FUNCTION_BLOCK FB_SL3K4
VAR CONSTANT
    nActiveMotorCount    : UINT := 4;
END_VAR
VAR_IN_OUT
	astMotionStage   : ARRAY[1..MotionConstants.MAX_STATE_MOTORS] OF ST_MotionStage;
	astChanParam     : ARRAY[1..MotionConstants.MAX_STATE_MOTORS] OF ST_MCS2ChanParameter;
    fbArbiter        : FB_Arbiter;
    fbFFHWO          : FB_HardwareFFOutput;
END_VAR
VAR_INPUT
	{attribute 'hide'}
    bFileReaderBusy      : BOOL;
	{attribute 'hide'}
    bFileReaderError     : BOOL;
	{attribute 'hide'}
    sTransitionKey       : STRING;
	{attribute 'hide'}
    bEnableDriftCheck    : BOOL := TRUE;
	{attribute 'hide'}
    fDriftTolerance      : LREAL := 0.003;
	{attribute 'hide'}
    bEnableBeamParams    : BOOL := TRUE;
    bReadDBNow           : BOOL;

END_VAR
VAR
    {attribute 'hide'}
    fbPerMotorFFO        : FB_PerMotorFFOND;
    {attribute 'hide'}
    fbMiscStatesErrorFFO : FB_MiscStatesErrorFFO;
    {attribute 'hide'}
    ffDriftFFO           : FB_FastFault;
    {attribute 'hide'}
    ffProgrammerError    : FB_FastFault;
    {attribute 'hide'}
    fbSL3K4BPTM          : FB_SL3K4BPTM;
    {attribute 'hide'}
    fbMotionClearAsserts : FB_MotionClearAsserts;
	
    {attribute 'pytmc' := '
        pv: STATE
        io: io
        field: DESC SL3K4 state
    '}
    eSL3K4State	: UINT := E_SL3K4State.NORMAL;
	
    {attribute 'pytmc' := 'pv: STATE'}
    stPMPSEpicsToPlc     : ST_StatePMPSEpicsToPlc;
	
    {attribute 'hide'}
    ePrevState            : E_SL3K4State := E_SL3K4State.NORMAL;

    {attribute 'hide'}
    abBladeEnable        : ARRAY[1..MotionConstants.MAX_STATE_MOTORS] OF BOOL;
    {attribute 'hide'}
    stMaintenanceGoal    : ST_DbStateParams;
    {attribute 'hide'}
    stNormalGoal         : ST_DbStateParams;
    {attribute 'hide'}
    stTransitionGoal     : ST_DbStateParams;
    {attribute 'hide'}
    bDBStatesLoaded      : BOOL := FALSE;
    {attribute 'hide'}
    bSafeToMove          : BOOL;
    {attribute 'hide'}
    bLocked              : BOOL;
    {attribute 'hide'}
    bMaintenanceActive   : BOOL;
    {attribute 'hide'}
    bProgrammerError     : BOOL;
    {attribute 'hide'}
    sStatusMsg           : STRING;
    {attribute 'hide'}
    bAnybladeError       : BOOL;
    {attribute 'hide'}
    bArbiterError        : BOOL;
    {attribute 'hide'}
    nBlades              : UINT;
    {attribute 'hide'}
    fbSL3K4ReadPMPSDB    : FB_SL3K4ReadPMPSDB;
    {attribute 'hide'}
    sDeviceName          : STRING := 'SL3K4';
    {attribute 'hide'}
    stGoalParams         : ST_DbStateParams;
    {attribute 'hide'}
    stTransParams        : ST_DbStateParams;
    {attribute 'hide'}
    bDBReloadRequested   : BOOL := TRUE;
    {attribute 'hide'}
    bDBReloadNow         : BOOL;
    {attribute 'hide'}
    bReadNow             : BOOL;
    {attribute 'hide'}
    bDone                : BOOL;
    {attribute 'hide'}
    bDriftFF             : BOOL;
    {attribute 'hide'}
    bLastTransAuth       : BOOL;
    {attribute 'hide'}
    bEnable              : BOOL;
    {attribute 'hide'}
    tArbiterTimeout      : TIME := T#3s;
    {attribute 'hide'}
    bMoveOnArbiterTimeout: BOOL := TRUE;
    {attribute 'hide'}
    bResetBPTMTimeout    : BOOL;
    {attribute 'hide'}
    bRetry               : BOOL;
    {attribute 'hide'}
    bAtState             : BOOL;
    {attribute 'hide'}
    bInternalAuth        : BOOL;
    {attribute 'hide'}
    bArbiterTimeout      : BOOL;
    arfDrift               : ARRAY[1..nActiveMotorCount] OF LREAL;
    {attribute 'hide'}
    allAxesIdle          : BOOL;
    {attribute 'hide'}
    axis                 : INT;
    {attribute 'hide'}
    i                    : DINT;
    {attribute 'hide'}
    bIsMaintenance       : BOOL;
    {attribute 'hide'}
    bGoalIsNormal        : BOOL;
    {attribute 'hide'}
    bFoundTransition     : BOOL;
    {attribute 'hide'}
    bFoundGoal           : BOOL;
    {attribute 'hide'}
    fbLogger             : FB_LogMessage := (eSubsystem:=E_SubSystem.MOTION);
    {attribute 'hide'}
    eSevr                : LCLS_General.TcEventSeverity;
    {attribute 'hide'}
    sLastStatusMsg       : STRING := '';
    {attribute 'hide'}
    eLastSevr            : TcEventSeverity := TcEventSeverity.Info;
    {attribute 'hide'}
    bTransitionAuthorized: BOOL;
    {attribute 'hide'}
    rtEnable             : R_TRIG;
    {attribute 'hide'}
    nGoalAtClear         : UINT;
    {attribute 'hide'}
    rtUpdateDBState      : R_TRIG;
    {attribute 'hide'}
    bFoundNormal         : BOOL;
    {attribute 'hide'}
    bFoundMaintenance    : BOOL;
	
    {attribute 'hide'}
    stDbStateParams      : ST_DbStateParams;
    {attribute 'hide'}
    bIsNormal: BOOL;
	{attribute 'hide'}
    rtTransAuth          : R_TRIG;
    {attribute 'hide'}
    rtTransDone          : R_TRIG;
    {attribute 'hide'}
    bModeTransitionStarted : BOOL;
    {attribute 'hide'}
    bModeTransitionDone : BOOL;
    {attribute 'hide'}
    bTransitionCompleted   : BOOL;
END_VAR



// --- PMPS DB Read / safety check (with reload logic) ---
fbSL3K4ReadPMPSDB(
    fbFFHWO := fbFFHWO,
    bFileReaderError := bFileReaderError,
    bFileReaderBusy  := bFileReaderBusy,
    sDeviceName      := sDeviceName,
    sTransitionKey   := sTransitionKey,
    jsonDoc          := PMPS_GVL.BP_jsonDoc,
    bReadDBNow :=bReadDBNow
);

// --- Early lock and fail-safe if DB not loaded ---
IF NOT fbSL3K4ReadPMPSDB.bStatesReady THEN
    FOR nBlades := 1 TO nActiveMotorCount DO
        astMotionStage[nBlades].bSafetyReady := FALSE;
        astChanParam[nBlades].bOverrideDirEnable := FALSE;
        abBladeEnable[nBlades] := FALSE;
    END_FOR
    bSafeToMove   := FALSE;
    bLocked       := TRUE;
    sStatusMsg    := 'PMPS parameter DB not loaded. Axes locked!';
    RETURN;
END_IF

// --- One-time extraction of DB states on rising edge ---
rtUpdateDBState(CLK := fbSL3K4ReadPMPSDB.bStatesReady);

IF rtUpdateDBState.Q THEN
    bFoundTransition := FALSE;
    bFoundNormal := FALSE;
    bFoundMaintenance := FALSE;

    FOR i := 0 TO UPPER_BOUND(fbSL3K4ReadPMPSDB.astDbStateParams, 1) DO
        IF fbSL3K4ReadPMPSDB.astDbStateParams[i].sPmpsState = sTransitionKey THEN
            stTransitionGoal := fbSL3K4ReadPMPSDB.astDbStateParams[i];
            bFoundTransition := TRUE;
        ELSIF fbSL3K4ReadPMPSDB.astDbStateParams[i].sPmpsState = 'SL3K4-MAINTENANCE' THEN
            stMaintenanceGoal := fbSL3K4ReadPMPSDB.astDbStateParams[i];
            bFoundMaintenance := TRUE;
        ELSIF fbSL3K4ReadPMPSDB.astDbStateParams[i].sPmpsState = 'SL3K4-NORMAL' THEN
                stNormalGoal := fbSL3K4ReadPMPSDB.astDbStateParams[i];
                bFoundNormal := TRUE;
        END_IF
    END_FOR

    IF NOT (bFoundTransition AND bFoundNormal AND bFoundMaintenance) THEN
        sStatusMsg := 'Error: Required PMPS state not found in DB!';
        bProgrammerError := TRUE;
    ELSE
        bDBStatesLoaded := TRUE;
    END_IF
END_IF
// 
IF bDBStatesLoaded THEN
    CASE eSL3K4State OF
        E_SL3K4State.MAINTENANCE: stGoalParams := stMaintenanceGoal;
        E_SL3K4State.NORMAL:      stGoalParams := stNormalGoal;
        ELSE                     stGoalParams := stNormalGoal; // Default fallback
    END_CASE
    stTransParams := stTransitionGoal;
END_IF

// --- Programmer error faulting ---
ffProgrammerError(
    i_xOK := NOT bProgrammerError,
    i_xAutoReset := TRUE,
    i_DevName := sDeviceName,
    i_Desc := 'Required PMPS state not found in DB or config error',
    i_TypeCode := E_MotionFFType.INTERNAL_ERROR,
    io_fbFFHWO := fbFFHWO
);

// --- Enable only if valid state/request, no errors ---
bEnable := ((eSL3K4State = E_SL3K4State.MAINTENANCE) OR (eSL3K4State = E_SL3K4State.NORMAL))
              AND NOT bProgrammerError
              AND stPMPSEpicsToPlc.bArbiterEnabled
              AND bEnableBeamParams;
rtEnable(CLK := bEnable);

// --- Aggregate blade errors ---
bAnybladeError := FALSE;
FOR nBlades := 1 TO nActiveMotorCount DO
    IF astMotionStage[nBlades].bError THEN
        bAnybladeError := TRUE;
    END_IF
END_FOR


// --- BPTM function block call ---
fbSL3K4BPTM(
    fbArbiter     := fbArbiter,
    fbFFHWO       := fbFFHWO,
    sDeviceName   := sDeviceName,
    stGoalParams  := stGoalParams,
    stTransParams := stTransParams,
    bEnable       := bEnable,
    bRetry        := rtEnable.Q AND nGoalAtClear = eSL3K4State,
    bBladeError   := bAnybladeError,
    bTransitionAuthorized => bTransitionAuthorized
);

// --- Clear asserts if BPTM not enabled ---
fbMotionClearAsserts(
    astDbStateParams := fbSL3K4ReadPMPSDB.astDbStateParams,
    fbArbiter        := fbArbiter,
    bExecute         := NOT fbSL3K4BPTM.bEnable
);

IF fbMotionClearAsserts.bExecute THEN
    nGoalAtClear := eSL3K4State;
END_IF

// Rising edge detection
rtTransAuth(CLK := bTransitionAuthorized);
rtTransDone(CLK := fbSL3K4BPTM.bDone);

// (reset only on mode change or BPTM error/busy)
IF rtTransAuth.Q THEN
    bModeTransitionStarted := TRUE;
END_IF
IF rtTransDone.Q THEN
    bModeTransitionDone := TRUE;
END_IF
bTransitionCompleted := bModeTransitionStarted AND bModeTransitionDone;

// Clear all transition flags & safe-to-move if a request starts or error/busy encountered
IF (eSL3K4State <> nGoalAtClear) OR fbSL3K4BPTM.bBusy OR fbSL3K4BPTM.bError THEN
    bSafeToMove := FALSE;
    bModeTransitionStarted := fbSL3K4BPTM.bBusy;
    bModeTransitionDone := FALSE;
    bTransitionCompleted := FALSE;
    nGoalAtClear := eSL3K4State;
END_IF

// --- Safe-to-Move calculation ---
CASE eSL3K4State OF
    E_SL3K4State.MAINTENANCE:
        bSafeToMove := bTransitionCompleted AND NOT bAnybladeError;
    E_SL3K4State.NORMAL:
        bSafeToMove := FALSE; // No motion in normal, just protection
    ELSE
        bSafeToMove := FALSE;
END_CASE
bLocked := NOT bSafeToMove;

// --- Per-blade enable/disable and drift detection ---
bDriftFF := FALSE;
FOR nBlades := 1 TO nActiveMotorCount DO
    CASE eSL3K4State OF
        E_SL3K4State.NORMAL:
            // disabled all blades
            abBladeEnable[nBlades] := FALSE;
            astMotionStage[nBlades].bSafetyReady := FALSE;
            astChanParam[nBlades].bOverrideDirEnable := FALSE;
			//beam parameters asserted?
            IF bTransitionCompleted THEN
                IF bEnableDriftCheck THEN
                    arfDrift[nBlades] := ABS(astMotionStage[nBlades].axis.NcToPlc.ActPos - astChanParam[nBlades].fPosition);
                    IF arfDrift[nBlades] > fDriftTolerance THEN
                        bDriftFF := TRUE;
                        // use  the drifttolerance in the error message.
                        sStatusMsg := CONCAT(astMotionStage[nBlades].sName, CONCAT('drifted out by', LREAL_TO_FMTSTR(arfDrift[nBlades],5,TRUE)));
                        astMotionStage[nBlades].sCustomErrorMessage := sStatusMsg;
                    END_IF
                END_IF
            END_IF
        E_SL3K4State.MAINTENANCE:
               astMotionStage[nBlades].bSafetyReady := FALSE;
            astChanParam[nBlades].bOverrideDirEnable := FALSE;
             abBladeEnable[nBlades] := FALSE;
            IF bSafeToMove THEN
                astMotionStage[nBlades].bSafetyReady := TRUE;
                astChanParam[nBlades].bOverrideDirEnable := TRUE;
                abBladeEnable[nBlades] := TRUE;
            END_IF
        ELSE
            astMotionStage[nBlades].bSafetyReady := FALSE;
            astChanParam[nBlades].bOverrideDirEnable := FALSE;
            abBladeEnable[nBlades] := FALSE;
    END_CASE
END_FOR

// --- Beam parameter feedback to error FB ---
IF bEnableBeamParams AND bDBStatesLoaded THEN
    fbMiscStatesErrorFFO.stCurrentBeamReq := stGoalParams.stBeamParams;
ELSE
    fbMiscStatesErrorFFO.stCurrentBeamReq := PMPS_GVL.cstFullBeam;
END_IF

fbMiscStatesErrorFFO(
    fbArbiter    := fbArbiter,
    fbFFHWO      := fbFFHWO,
    sDeviceName  := sDeviceName,
    bKnownState  := eSL3K4State > 0,
    nTransitionID:= stTransParams.nRequestAssertionID
);

// --- Per-motor fast fault & drift fault FBs ---
fbPerMotorFFO(
    astMotionStage     := astMotionStage,
    fbFFHWO            := fbFFHWO,
    nActiveMotorCount  := nActiveMotorCount,
    sDeviceName        := sDeviceName
);

ffDriftFFO(
    i_xOK        := NOT bDriftFF,
    i_xAutoReset := TRUE,
    i_DevName    := sDeviceName,
    i_Desc       := 'Blades drifted beyond allowable delta',
    i_TypeCode   := E_MotionFFType.INTERNAL_ERROR,
    io_fbFFHWO   := fbFFHWO
);

// --- Status message and logging ---
IF bDriftFF OR bProgrammerError THEN
    sStatusMsg := 'Device fast faulted (blades, encoder, or config error)';
    eSevr := TcEventSeverity.Critical;
ELSIF bSafeToMove THEN
    sStatusMsg := 'Maintenance: PMPS safe, axes enabled for manual scatter/homing.';
    eSevr := TcEventSeverity.Info;
ELSE
    IF (eSL3K4State = E_SL3K4State.NORMAL) THEN
        sStatusMsg := 'Normal: Axes locked for PMPS protection.';
        eSevr := TcEventSeverity.Info;
    ELSE
        sStatusMsg := 'Axes locked in undefined or error state.';
        eSevr := TcEventSeverity.Warning;
    END_IF
END_IF

// --- Log only on change ---
IF (sStatusMsg <> sLastStatusMsg) THEN
    fbLogger(
        sMsg  := sStatusMsg,
        eSevr := eSevr
    );
    sLastStatusMsg := sStatusMsg;
    eLastSevr := eSevr;
END_IF

END_FUNCTION_BLOCK

(* stored: Version 1.1.0.1
   POU FB_SL3K4: Id {dec1d628-e499-461c-bd3b-fc39c76517dd}, SpecialFunc None *)
